(* LS Electric XG5000 project: 클레이사격 *)
(* PLC LSPLC *)

FUNCTION_BLOCK Randomize
(* 랜덤을 만드는 기능이다. *)
VAR_INPUT
    INPUT : BOOL;
END_VAR
VAR_OUTPUT
    RESULT : UDINT;
END_VAR
VAR
    OUT : UDINT;
    게임시작 : BOOL;
    업카운터 : CTU_UINT;
END_VAR

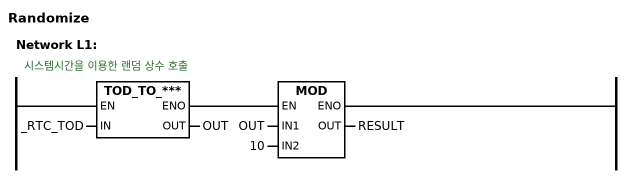
(* 시스템시간을 이용한 랜덤 상수 호출 *)
(* Rung L1 *)
OUT := TOD_TO_***(_RTC_TOD);
RESULT := OUT MOD 10;
END_FUNCTION_BLOCK

PROGRAM 1namal (* task: 스캔 프로그램 *)
VAR
    ET : TIME;
    INPUT : BOOL;
    INST : TRTG;
    INST1 : TRTG;
    MODE : USINT;
    OUT : STRING;
    PV : UINT;
    R : BOOL;
    R2S : STRING;
    RandTime : STRING;
    RESULT : UDINT;
    RST : BOOL;
    SEC : INT;
    zmf0 : BOOL;
    게임시간 : TRTG;
    게임시작 AT %IX0.0.0 : BOOL;
    게임중 AT %QX0.1.22 : BOOL;
    남은 : BOOL;
    남은탄약 AT %QW0.3.0 : UINT;
    도착전1 : TON;
    득점 : BOOL;
    딜레이 : TOF;
    랜덤상수 : Randomize;
    명중 : BOOL;
    명중0 : BOOL;
    명중1 : BOOL;
    명중2 : BOOL;
    명중3 : BOOL;
    명중4 : BOOL;
    명중5 : BOOL;
    명중6 : BOOL;
    명중7 : BOOL;
    명중8 : BOOL;
    명중9 : BOOL;
    명중시간0 : TP;
    명중시간1 : TP;
    명중시간2 : TP;
    명중시간3 : TP;
    명중시간4 : TP;
    명중시간5 : TP;
    명중시간6 : TP;
    명중시간7 : TP;
    명중시간8 : TP;
    명중시간9 : TP;
    명중전 : TIME;
    명중전0 : TON;
    명중전1 : TON;
    명중전2 : TON;
    명중전3 : TON;
    명중전4 : TON;
    명중전5 : TON;
    명중전6 : TON;
    명중전7 : TON;
    명중전8 : TON;
    명중전9 : TON;
    비행시간 : TIME;
    비행시간0 : TRTG;
    비행시간1 : TRTG;
    비행시간2 : TRTG;
    비행시간3 : TRTG;
    비행시간4 : TRTG;
    비행시간5 : TRTG;
    비행시간6 : TRTG;
    비행시간7 : TRTG;
    비행시간8 : TRTG;
    비행시간9 : TRTG;
    시간 AT %QW0.3.2 : INT;
    시간1 : TRTG;
    시간나누기 : TIME_DE;
    오른쪽사격 AT %IX0.0.2 : BOOL;
    왼쪽사격 AT %IX0.0.1 : BOOL;
    장전속도 : TON;
    재장전 AT %QX0.1.5 : BOOL;
    재장전버튼 AT %IX0.0.3 : BOOL;
    적중시간 : TIME;
    점수 AT %QW0.3.1 : UINT;
    점수판 : CTU_UINT;
    총격파티클_오른쪽 AT %QX0.1.3 : BOOL;
    총격파티클_왼쪽 AT %QX0.1.2 : BOOL;
    총구방향_오른쪽 AT %QX0.1.1 : BOOL;
    총구방향_왼쪽 AT %QX0.1.0 : BOOL;
    총알카운트 : CTD_UINT;
    클0 AT %QX0.1.10 : BOOL;
    클1 AT %QX0.1.11 : BOOL;
    클2 AT %QX0.1.12 : BOOL;
    클3 AT %QX0.1.13 : BOOL;
    클4 AT %QX0.1.14 : BOOL;
    클5 AT %QX0.1.15 : BOOL;
    클6 AT %QX0.1.16 : BOOL;
    클7 AT %QX0.1.17 : BOOL;
    클8 AT %QX0.1.18 : BOOL;
    클9 AT %QX0.1.19 : BOOL;
    클레이0 : BOOL;
    클레이1 : BOOL;
    클레이2 : BOOL;
    클레이3 : BOOL;
    클레이4 : BOOL;
    클레이5 : BOOL;
    클레이6 : BOOL;
    클레이7 : BOOL;
    클레이8 : BOOL;
    클레이9 : BOOL;
    클레이던지기 : TIME;
    탄약1 AT %QX0.1.20 : BOOL;
    탄약2 AT %QX0.1.21 : BOOL;
    플라이클레이 : TOF;
    확인 : BOOL;
END_VAR
VAR
    _e1 : R_TRIG;
    _e2 : R_TRIG;
    _t3 : BOOL;
    _e4 : R_TRIG;
END_VAR

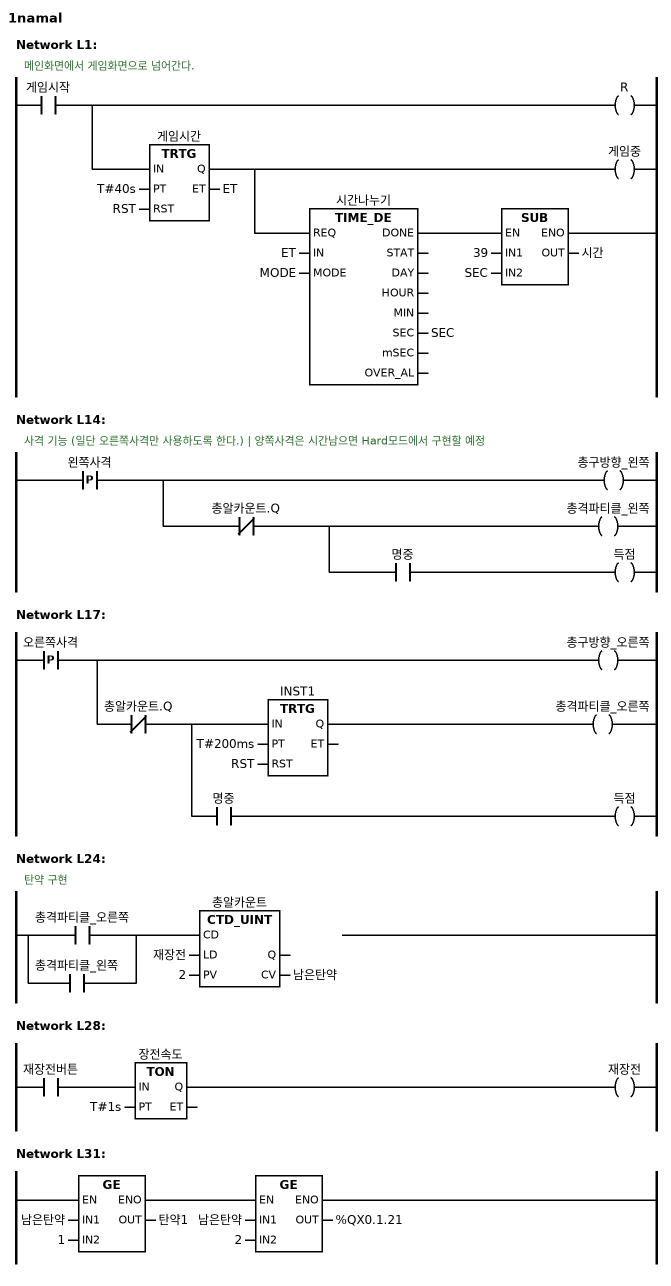
(* 메인화면에서 게임화면으로 넘어간다. *)
(* Rung L1 *)
R := 게임시작;
게임시간(IN := 게임시작, PT := T#40s, RST := RST, ET => ET);
게임중 := 게임시간.Q;
시간나누기(REQ := 게임시간.Q, IN := ET, MODE := MODE, SEC => SEC);
IF 시간나누기.DONE THEN 시간 := 39 - SEC; END_IF;
(* 사격 기능 (일단 오른쪽사격만 사용하도록 한다.) | 양쪽사격은 시간남으면 Hard모드에서 구현할 예정 *)
(* Rung L14 *)
_e1(CLK := 왼쪽사격);
총구방향_왼쪽 := _e1.Q;
총격파티클_왼쪽 := _e1.Q AND NOT 총알카운트.Q;
득점 := _e1.Q AND NOT 총알카운트.Q AND 명중;
(* Rung L17 *)
_e2(CLK := 오른쪽사격);
총구방향_오른쪽 := _e2.Q;
INST1(IN := _e2.Q AND NOT 총알카운트.Q, PT := T#200ms, RST := RST);
총격파티클_오른쪽 := INST1.Q;
득점 := _e2.Q AND NOT 총알카운트.Q AND 명중;
(* 탄약 구현 *)
(* Rung L24 *)
총알카운트(CD := 총격파티클_오른쪽 OR 총격파티클_왼쪽, LD := 재장전, PV := 2, CV => 남은탄약);
(* Rung L28 *)
장전속도(IN := 재장전버튼, PT := T#1s);
재장전 := 장전속도.Q;
(* Rung L31 *)
탄약1 := 남은탄약 >= 1;
%QX0.1.21 := 남은탄약 >= 2;

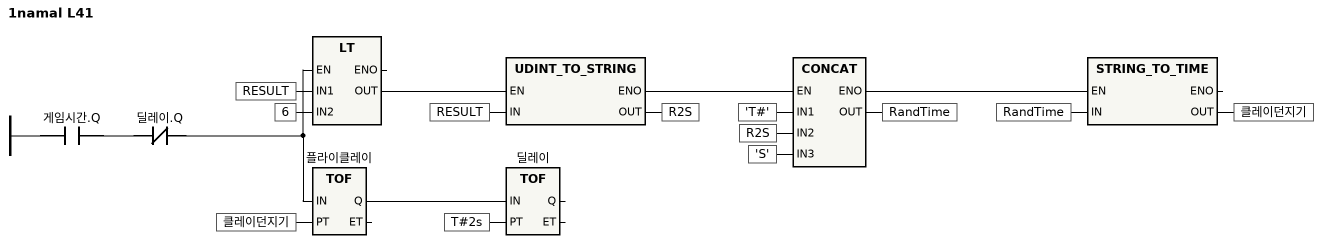
(* 클레이(접시)가 던져지는 타이밍 기능 *)
(* Rung L41 *)
IF 게임시간.Q AND NOT 딜레이.Q THEN _t3 := RESULT < 6; END_IF;
IF _t3 THEN
    R2S := UDINT_TO_STRING(RESULT);
    RandTime := CONCAT('T#', R2S, 'S');
    클레이던지기 := STRING_TO_TIME(RandTime);
END_IF;
플라이클레이(IN := 게임시간.Q AND NOT 딜레이.Q, PT := 클레이던지기);
딜레이(IN := 플라이클레이.Q, PT := T#2s);

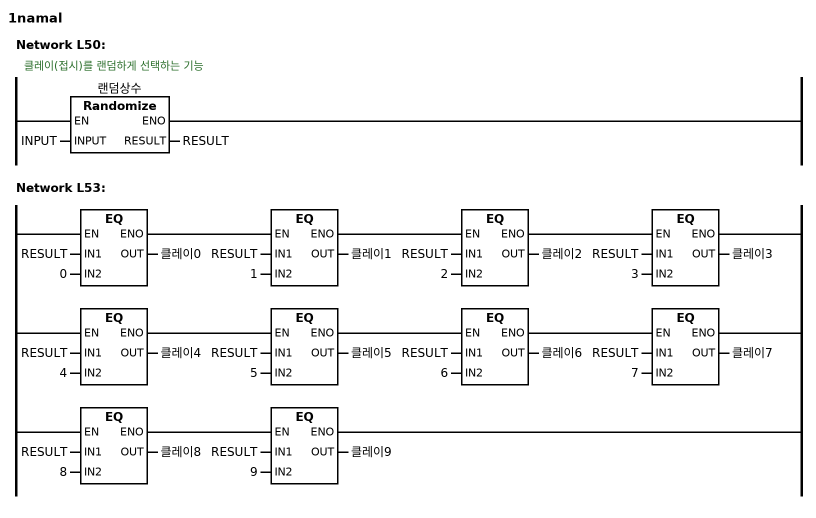
(* 클레이(접시)를 랜덤하게 선택하는 기능 *)
(* Rung L50 *)
랜덤상수(INPUT := INPUT, RESULT => RESULT);
(* Rung L53 *)
클레이0 := RESULT = 0;
클레이1 := RESULT = 1;
클레이2 := RESULT = 2;
클레이3 := RESULT = 3;
클레이4 := RESULT = 4;
클레이5 := RESULT = 5;
클레이6 := RESULT = 6;
클레이7 := RESULT = 7;
클레이8 := RESULT = 8;
클레이9 := RESULT = 9;

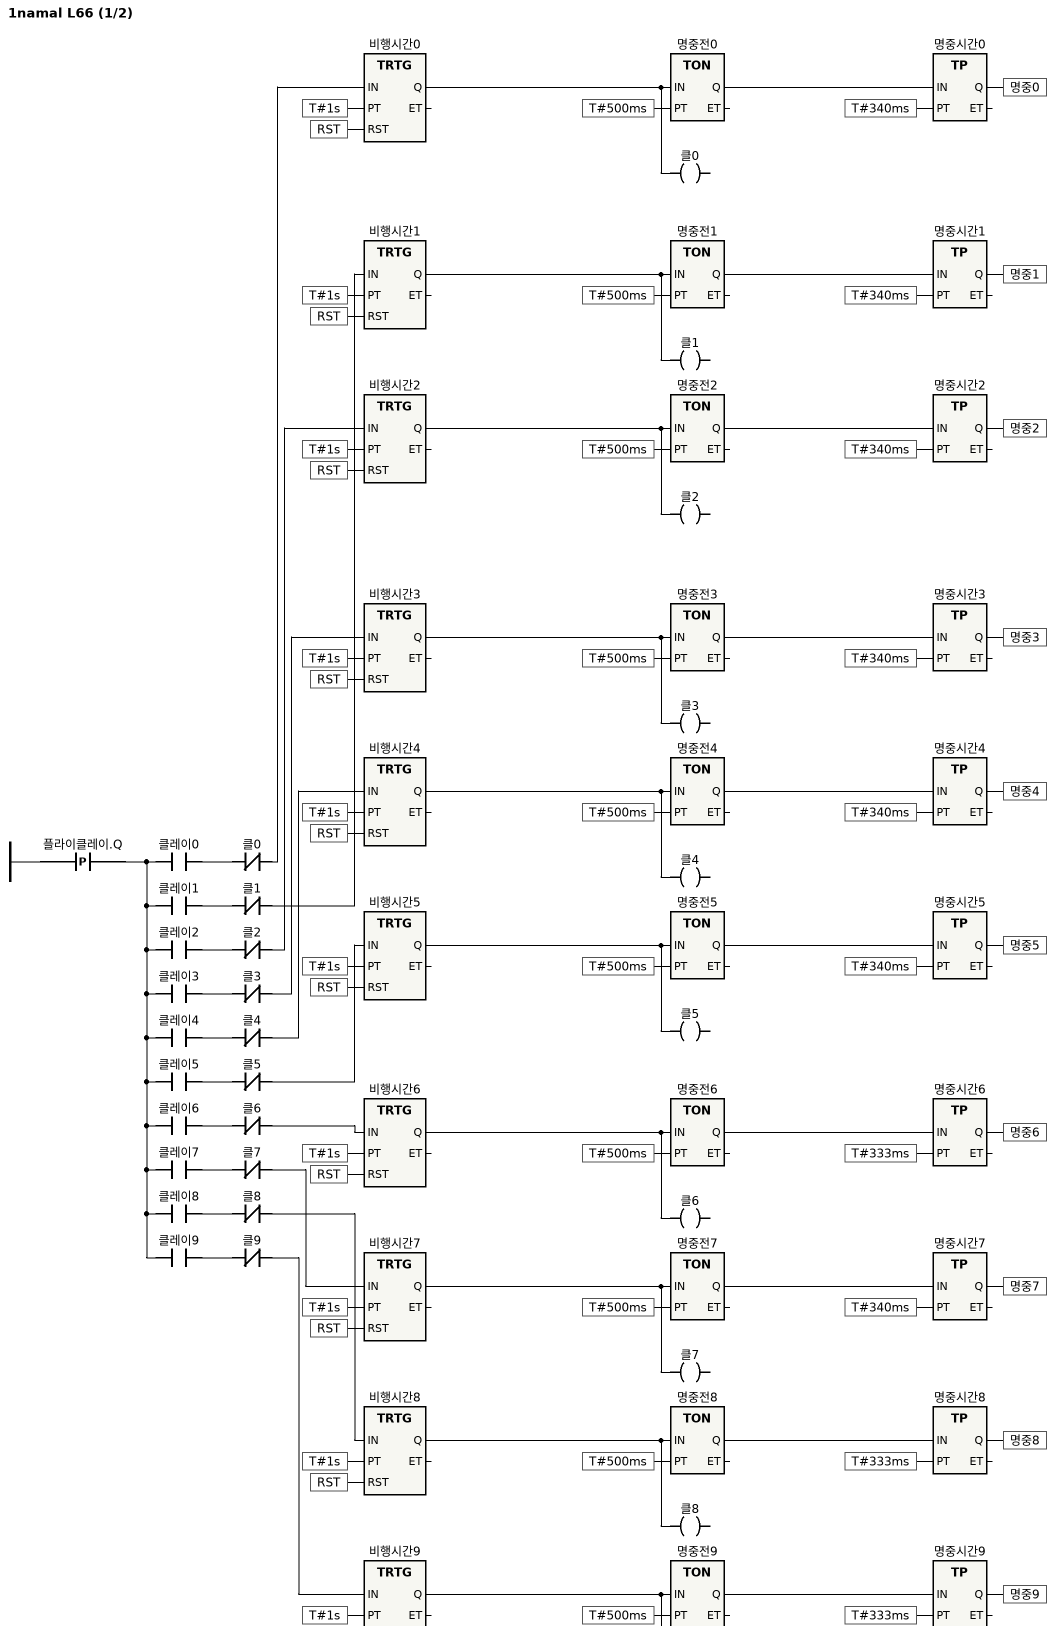

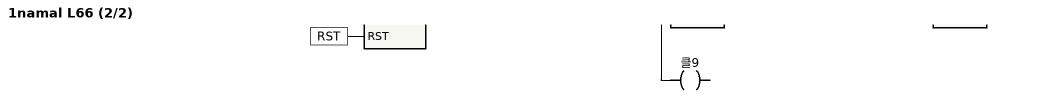
(* 각 클레이(접시)마다 속도 *)
(* Rung L66 *)
_e4(CLK := 플라이클레이.Q);
비행시간0(IN := _e4.Q AND 클레이0 AND NOT 클0, PT := T#1s, RST := RST);
클0 := 비행시간0.Q;
명중전0(IN := 비행시간0.Q, PT := T#500ms);
명중시간0(IN := 명중전0.Q, PT := T#340ms);
명중0 := 명중시간0.Q;
비행시간1(IN := _e4.Q AND 클레이1 AND NOT 클1, PT := T#1s, RST := RST);
클1 := 비행시간1.Q;
명중전1(IN := 비행시간1.Q, PT := T#500ms);
명중시간1(IN := 명중전1.Q, PT := T#340ms);
명중1 := 명중시간1.Q;
비행시간2(IN := _e4.Q AND 클레이2 AND NOT 클2, PT := T#1s, RST := RST);
클2 := 비행시간2.Q;
명중전2(IN := 비행시간2.Q, PT := T#500ms);
명중시간2(IN := 명중전2.Q, PT := T#340ms);
명중2 := 명중시간2.Q;
비행시간3(IN := _e4.Q AND 클레이3 AND NOT 클3, PT := T#1s, RST := RST);
클3 := 비행시간3.Q;
명중전3(IN := 비행시간3.Q, PT := T#500ms);
명중시간3(IN := 명중전3.Q, PT := T#340ms);
명중3 := 명중시간3.Q;
비행시간4(IN := _e4.Q AND 클레이4 AND NOT 클4, PT := T#1s, RST := RST);
클4 := 비행시간4.Q;
명중전4(IN := 비행시간4.Q, PT := T#500ms);
명중시간4(IN := 명중전4.Q, PT := T#340ms);
명중4 := 명중시간4.Q;
비행시간5(IN := _e4.Q AND 클레이5 AND NOT 클5, PT := T#1s, RST := RST);
클5 := 비행시간5.Q;
명중전5(IN := 비행시간5.Q, PT := T#500ms);
명중시간5(IN := 명중전5.Q, PT := T#340ms);
명중5 := 명중시간5.Q;
비행시간6(IN := _e4.Q AND 클레이6 AND NOT 클6, PT := T#1s, RST := RST);
클6 := 비행시간6.Q;
명중전6(IN := 비행시간6.Q, PT := T#500ms);
명중시간6(IN := 명중전6.Q, PT := T#333ms);
명중6 := 명중시간6.Q;
비행시간7(IN := _e4.Q AND 클레이7 AND NOT 클7, PT := T#1s, RST := RST);
클7 := 비행시간7.Q;
명중전7(IN := 비행시간7.Q, PT := T#500ms);
명중시간7(IN := 명중전7.Q, PT := T#340ms);
명중7 := 명중시간7.Q;
비행시간8(IN := _e4.Q AND 클레이8 AND NOT 클8, PT := T#1s, RST := RST);
클8 := 비행시간8.Q;
명중전8(IN := 비행시간8.Q, PT := T#500ms);
명중시간8(IN := 명중전8.Q, PT := T#333ms);
명중8 := 명중시간8.Q;
비행시간9(IN := _e4.Q AND 클레이9 AND NOT 클9, PT := T#1s, RST := RST);
클9 := 비행시간9.Q;
명중전9(IN := 비행시간9.Q, PT := T#500ms);
명중시간9(IN := 명중전9.Q, PT := T#333ms);
명중9 := 명중시간9.Q;

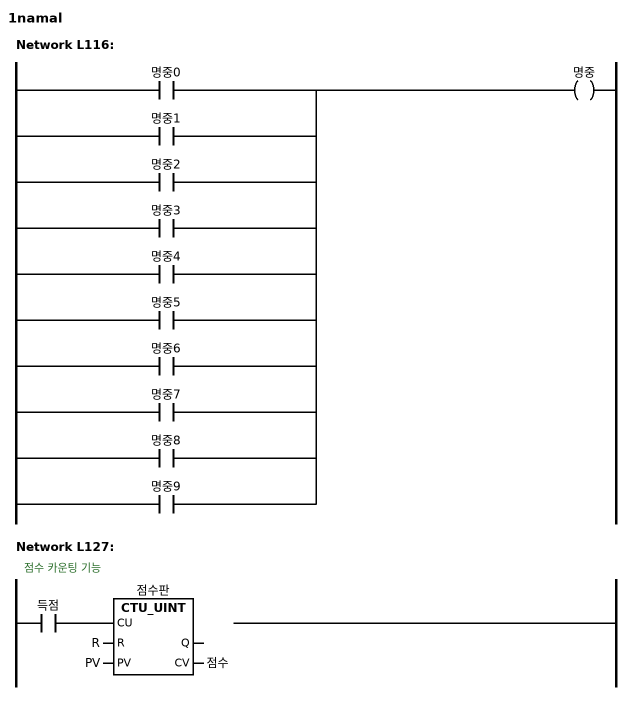
(* Rung L116 *)
명중 := 명중0 OR 명중1 OR 명중2 OR 명중3 OR 명중4 OR 명중5 OR 명중6 OR 명중7 OR 명중8 OR 명중9;
(* 점수 카운팅 기능 *)
(* Rung L127 *)
점수판(CU := 득점, R := R, PV := PV, CV => 점수);
END_PROGRAM